    |       background_ready = 0
    |       global move_p = background_pose
    |       wv_wp2 = th_wv_wp2
    |       if(par_2f):
    |         background_cal=1
    |       else:
    |         background_cal=1
    |       end
    |       global a_val = 3
    |       if(a_val >= 30):
    |         write_port_register(142,112)
    |         sleep(0.5)
    |         halt
    |       end
    |     end
    | 
    |     if(wv_weldpar[5] ==1):
    |         if( (sin_dir==1 and wving_delay[0]==0) or (sin_dir==-1 and wving_delay[2]==0)):
    |          tri_count = tri_count + 1
    |         end
    |         global target_p = move_p[tri_count]
    |         target_p=p[target_p[0],target_p[1],target_p[2],target_p[3],target_p[4],target_p[5]]
    |         tri_count = tri_count + 1
    |     elif(wv_weldpar[5] ==2):
    |       if( (tri_count==1 and sin_dir==1 and wving_delay[0]==0) or (tri_count==1 and sin_dir==-1 and wving_delay[2]==0)):
    |        tri_count = tri_count + 1
    |       end
    |       global target_p = move_p[tri_count]
    |       target_p=p[target_p[0],target_p[1],target_p[2],target_p[3],target_p[4],target_p[5]]
    |       tri_count = tri_count + 1
    |     else:
    |       popup("Please insert 0 - sin or 1 - triangle")
    |     end
    |     if(target_p == p[0,0,0,0,0,0]):
    |       target_p = get_actual_tcp_pose()
    |     end
    |     # write_output_float_register(25,tri_count)
    |     if((norm(tri_count)== 1) and sin_dir==1 and wving_delay[0]>0):
    |       movel(target_p,a=a_val,v=wv_system_speed/1000)
    |       peak_value = 0
    |       sleep(wving_delay[0])
    |       peak_value = 100
    |     elif((norm(tri_count)== 2) and sin_dir==1 and wving_delay[1]>0):
    |       movel(target_p,a=a_val,v=wv_system_speed/1000)
    |       peak_value = 0
    |       sleep(wving_delay[1])
    |       peak_value = 100
    |     elif((norm(tri_count)== 1) and sin_dir==-1 and wving_delay[2]>0):
    |       movel(target_p,a=a_val,v=wv_system_speed/1000)
    |       peak_value = 0
    |       sleep(wving_delay[2])
    |       peak_value = 100
    |     elif((norm(tri_count)== 2) and sin_dir==-1 and wving_delay[3]>0):
    |       movel(target_p,a=a_val,v=wv_system_speed/1000)
    |       peak_value = 0
    |       sleep(wving_delay[3])
    |       peak_value = 100
    |     else:
    |       movel(target_p,a=a_val,v=wv_system_speed/1000)
    |       peak_value = 100
    |     end
    |     global last_pose = target_p
    |   end
    |   timer_1_is_counting = False
    | 
    |   if(a9_wv_weldingon == True and wving_crater[5]!=0):
    |     #crater end option
    |     set_current_voltage(wving_crater[3],wving_crater[4])
    |     sleep(wving_crater[5])
    |     program_weld_on = False
    |     set_current_voltage(ext_fun[1],ext_fun[0])
    |     if(isHicomm):
    |       write_port_register(202,0)
    |       write_port_register(149,0)
    |     else:
    |       set_standard_digital_out(0,False)
    |     end
    |     while(read_welder(5)==True):
    |       if(weld_onoff==True):
    |         write_welder(0,False)
    |       end
    |       sync()
    |     end
    |   end
    |   timer_counter = 0
    |   kill CThread
    |   kill DThread
    |   kill TThread
    |   timer_counter = 0
    |   timer_counting = False
    |   wcr_counter = 0
    |   wcr_counting = False
    |   get_wcr = False
    |   welding_off_t = 0
    | 
    |   if(wv_seq[0] == 0 or wv_seq[0] == 3):
    |     if(a9_wv_weldingon==True):
    |       program_weld_on = False
    |       write_port_register(202,0)
    |       write_port_register(149,0)
    |       write_welder(0,False)
    |       if(wv_weldpar[2]==1):
    |         target_pos = feature_offset(get_actual_tcp_pose(),p[0,0,-0.01,0,0,0],wv_Line_Feature2)
    |         movel(target_pos,0.5,0.01)
    |       end
    |     end
    |   end
    |   background_pose = [dumy_p,dumy_p,dumy_p]
    |   move_p = background_pose
    |   return sin_dir
    | end
    | 
    | 
    | def line_weaving_tp_l(wv_wp1,wv_wp3,wv_weldpar=[100,10,0,1,5,1,1],tilt_deg=[0,0,0],wving_delay=[0,0,0,0],welding_on=False,Arc_sen=[0,0,0,0,0,0],wv_gap=[0,0,0,0],z_param=[0,0,0,0,0],par_2f=False,wving_crater=[0,0,0,0,0,0,0,0,0,0],ext_fun=[0,0,0,0,0,0,0,0,0,0,0],wv_seq = [0,-1],wv_feature=p[0,0,0,0,0,0]):
    |   global start_gas_time = 2
    |   global counter_average = 1
    |   global counter_average_num = 0
    |   global waste_cycle = ext_fun[8]
    |   global current_list = 0
    |   global wv_wp4 = wv_wp3
    |   global A_T1 = wv_wp4[0]
    |   global A_T2 = wv_wp4[1]
    |   global A_T3 = wv_wp4[2]
    |   if(par_2f):
    |     global squash_cycle = 0
    |   else:
    |     global squash_cycle = ext_fun[7]
    |   end
    |   global th_ext_fun = ext_fun
    |   RTDE_init()
    | 
    |   if (wv_gap[0]==1):
    |     gap_check = True
    |     wv_gap[0]=0
    |   else:
    |     gap_check= False
    |   end
    |   # e-Series 2, CB-Seris 8
    |   global system_bus_ms = 2
    | 
    |   global sin_dir = wv_seq[1]
    |   global start_trig = False
    |   dir=1
    | 
    |   global tri_count=0
    | 
    |   global z_bottom = z_param[0]/1000
    |   if(wv_weldpar[6]==-1):
    |     global vir_v = -1
    |   else:
    |     global vir_v = 1
    |   end
    | 
    |   if(par_2f):
    |     global cal_off_ang_rx = 1
    |     global cal_off_ang_ry = 0
    |   else:
    |     global cal_off_ang_rx = 0
    |     global cal_off_ang_ry = 1
    |   end
    | 
    |   if(wv_seq[0] == 2 or wv_seq[0] == 3):
    |     tilt_deg = [0,0,0]
    |     global cal_off_ang_rx = 0
    |     global cal_off_ang_ry = 0
    |   end
    | 
    |   global wv_Line_Feature2 = wv_wp1
    |   if(wv_weldpar[0] > 700 and par_2f == False):
    |     wv_weldpar[0] = 700
    |   end
    |   if(wv_wp3[0]==p[0,0,0,0,0,0]):
    |     global wv_wp2 = feature_offset(wv_wp1,p[wv_weldpar[0]/1000,0,0,0,0,0],wv_Line_Feature2)
    |   else:
    |     global wv_wp2 = wv_wp4[0]
    |     wv_weldpar[0] = point_dist(wv_wp1,wv_wp2)*1000
    |     global wv_dist_bak = point_dist(wv_wp1,wv_wp2)*1000
    |   end
    |   if(wv_seq[0] == 2 or wv_seq[0] == 3):
    |     wv_Line_Feature2 = wv_feature
    |   end
    |   #setting
    |   if(par_2f):
    |     #todo - 1
    |     offset_2f_k = -1 * ext_fun[9]
    |     offset_2f_z = 1 * ext_fun[10]
    |     if(wv_seq[0] == 0 or wv_seq[0] == 1):
    |       line_feature = get_feature_Line(wv_wp1,wv_wp2)
    |       b_p1 = wv_wp1
    |       b_p2 = feature_offset(wv_wp1,p[0,0.01*vir_v,0,0,0,0],line_feature)
    |       b_p3 = pose_add(wv_wp1,p[0,0,0.01,0,0,0])
    | 
    |       back_feature = get_feature_plane_xz(b_p1,b_p2,b_p3)
    |       wv_wp1 = pose_trans(wv_wp1,p[0,0,0,0,0,d2r(-90)])
    |       wv_wp1 = feature_offset(wv_wp1,p[0,offset_2f_k/1000,0,0,0,0],back_feature)
    |       wv_wp1 = pose_add(wv_wp1,p[0,0,offset_2f_z/1000,0,0,0])
    |       # wv_wp1 = pose_add(wv_wp1,p[offset_2f_k/1000,0,0,0,0,0])
    |     end
    |       # wv_wp2 = pose_add(wv_wp2,p[offset_2f_k/1000,0,0,0,0,0])
    |       wv_wp2 = feature_offset(wv_wp2,p[0,offset_2f_k/1000,0,0,0,0],back_feature)
    |       wv_wp2 = pose_add(wv_wp2,p[0,0,offset_2f_z/1000,0,0,0])
    |       wv_wp2 = p[wv_wp2[0],wv_wp2[1],wv_wp2[2],wv_wp1[3],wv_wp1[4],wv_wp1[5]]
    | 
    |       wv_wp3_p = feature_offset(wv_wp3[0],p[0,offset_2f_k/1000,0,0,0,0],back_feature)
    |       wv_wp3_p = pose_add(wv_wp3_p,p[0,0,offset_2f_z/1000,0,0,0])
    |       wv_wp3_p = p[wv_wp3_p[0],wv_wp3_p[1],wv_wp3_p[2],wv_wp1[3],wv_wp1[4],wv_wp1[5]]
    |       wv_wp4[0] = p[wv_wp3_p[0],wv_wp3_p[1],wv_wp3_p[2],wv_wp1[3],wv_wp1[4],wv_wp1[5]]
    | 
    |       wv_wp3_p = feature_offset(wv_wp3[1],p[0,offset_2f_k/1000,0,0,0,0],back_feature)
    |       wv_wp3_p = pose_add(wv_wp3_p,p[0,0,offset_2f_z/1000,0,0,0])
    |       wv_wp3_p = p[wv_wp3_p[0],wv_wp3_p[1],wv_wp3_p[2],wv_wp1[3],wv_wp1[4],wv_wp1[5]]
    |       wv_wp4[1] = p[wv_wp3_p[0],wv_wp3_p[1],wv_wp3_p[2],wv_wp1[3],wv_wp1[4],wv_wp1[5]]
    | 
    |       wv_wp3_p = feature_offset(wv_wp3[2],p[0,offset_2f_k/1000,0,0,0,0],back_feature)
    |       wv_wp3_p = pose_add(wv_wp3_p,p[0,0,offset_2f_z/1000,0,0,0])
    |       wv_wp3_p = p[wv_wp3_p[0],wv_wp3_p[1],wv_wp3_p[2],wv_wp1[3],wv_wp1[4],wv_wp1[5]]
    |       wv_wp4[2] = p[wv_wp3_p[0],wv_wp3_p[1],wv_wp3_p[2],wv_wp1[3],wv_wp1[4],wv_wp1[5]]
    |   end
    |   if(ext_fun[2]==1 and par_2f==False):
    |     #squash
    |     w_voltage = ext_fun[3]
    |     w_current = ext_fun[4]
    |     set_current_voltage(w_current,w_voltage)
    |     global cir_speed_org_bak = wv_weldpar[1]
    |     global wving_amplitude_bak = wv_weldpar[4]
    |     wv_weldpar[1] = ext_fun[6]
    |     wv_weldpar[4] = ext_fun[5]
    |   end
    |   if(par_2f):
    |     global wv_system_speed = calculate_2f(wv_weldpar[4],wv_wp1,wv_wp2,wv_weldpar[1],wv_weldpar[3],wving_delay,wving_crater)
    |   else:
    |     global wv_system_speed = calculate_3f(wv_weldpar[4],wv_wp1,wv_wp2,wv_weldpar[1],wv_weldpar[3],wving_delay)
    |     x_radius = x_radius / 1000
    |   end
    |   global wv_set_speed = wv_system_speed
    |   ratio_t=0
    |   # mm -> m
    |   global y_radius = y_radius / 1000
    |   global y_radius_bak = y_radius
    |   #init for thread
    |   global ext_stick = 0
    |   global th_arc_sen=Arc_sen
    |   global th_wv_gap=wv_gap
    |   global th_tilt_deg=tilt_deg
    |   global last_tilt_deg =th_tilt_deg
    |   global last_wv_wp1 = wv_wp1
    |   global last_wv_line = wv_Line_Feature2
    |   global th_wving_crater=wving_crater
    |   global last_z_bottom = z_bottom
    |   global th_par_2f = par_2f
    |   global th_cir_speed_org=wv_weldpar[1]
    |   global th_wv_wp1 = wv_wp1
    |   global th_wv_wp2 = wv_wp2
    |   global th_wv_wp3 = wv_wp3[0]
    |   global th_wv_weldpar=wv_weldpar
    |   global th_wving_delay=wving_delay
    |   global th_z_param=z_param
    |   global th_wv_seq = wv_seq
    |   global th_wv_feature=wv_feature
    |   global th_dir = dir
    | 
    |   # if want to use approach position
    |   if(wv_seq[0] ==0 or wv_seq[0] == 1):
    |     global get_angle_rx = welding_angle_cal_2f(wv_wp1[1],tilt_deg,vir_v,cal_off_ang_rx)
    |     global get_angle_ry = welding_angle_cal_3f(wv_wp1[2],tilt_deg,z_bottom,cal_off_ang_ry)
    | 
    |     target_p = feature_offset(wv_wp1,p[0,0,0,d2r(tilt_deg[0] + get_angle_rx),d2r(tilt_deg[1] + get_angle_ry),d2r(tilt_deg[2])],wv_Line_Feature2)
    | 
    |     if(wv_weldpar[2]==1):
    |       target_p_appr = feature_offset(target_p,p[0,0,-0.02,0,0,0],wv_Line_Feature2)
    |       movel(target_p_appr,a=0.5,v=0.125)
    |     end
    |     movel(target_p,a=0.5,v=0.125)
    |   end
    | 
    |   CThread = run CalThread()
    |   DThread = run diff_Thread()
    |   TThread = run thread_timer()
    |   global timer_counting=True
    |   global program_weld_on = True
    | 
    |   if(a9_wv_weldingon==True):
    |     while(welding_off_t==55):
    |       sync()
    |     end
    |     if(wving_crater[2]>0):
    |       set_current_voltage(wving_crater[0],wving_crater[1])
    |     end
    |     if(welding_off_t != 1):
    |       write_welder(0,True)
    |       while(get_wcr==False):
    |         if(weld_onoff==False):
    |           write_welder(0,True)
    |         end
    |         sync()
    |       end
    |       if(wving_crater[2]>0):
    |         #Crater Begin option
    |         write_output_float_register(1,1)
    |         sleep(wving_crater[2])
    |         set_current_voltage(ext_fun[1],ext_fun[0])
    |       end
    |     end
    |   end
    |   start_gas_time = 0
    | 
    |   background_cal=1
    |   background_ready=0
    |   FT_trig=True
    | 
    |   timer_1_is_counting = True
    | 
    |   while((ratio_t < 1) or current_list==0 or current_list==1):
    |     if(ratio_t>=1 and current_list!=2):
    |       if (gap_check):
    |         gap_check = True
    |         wv_gap[0]=1
    |         th_wv_gap[0]=1
    |         gap_check= False
    |       end
    |       ratio_t=0
    |       if(current_list==0):
    |         wving_amp_bak = wv_weldpar[4]
    |         wv_weldpar[4] = wv_weldpar[4] * 1
    |         th_wv_weldpar[4] = wv_weldpar[4]
    |         circle_speed_bak = wv_weldpar[1]
    |         wv_weldpar[1]= wv_weldpar[1]*0.7
    |         th_wv_weldpar[1]= wv_weldpar[1]
    |       elif(current_list==1):
    |         wv_weldpar[4] = wving_amp_bak
    |         th_wv_weldpar[4] = wv_weldpar[4]
    |         wv_weldpar[1] = circle_speed_bak
    |         th_wv_weldpar[1]= wv_weldpar[1]
    |       end
    |       wv_wp1=wv_wp4[current_list]
    |       wv_wp2=wv_wp4[current_list+1]
    |       global th_wv_wp1 = wv_wp4[current_list]
    |       global th_wv_wp2 = wv_wp4[current_list+1]
    |       global th_wv_wp3 = wv_wp4[current_list+1]
    |       wv_system_speed_bak = wv_system_speed
    |       if(par_2f):
    |         global wv_system_speed = calculate_2f(wv_weldpar[4],wv_wp4[current_list],wv_wp4[current_list+1],wv_weldpar[1],wv_weldpar[3],wving_delay,wving_crater)
    |         global y_radius = y_radius / 1000
    |         global y_radius_bak = y_radius
    |       else:
    |         global wv_system_speed = calculate_3f(wv_weldpar[4],wv_wp4[current_list],wv_wp4[current_list+1],wv_weldpar[1],wv_weldpar[3],wving_delay)
    |         x_radius = x_radius / 1000
    |       end
    |       wv_system_speed = wv_system_speed_bak
    |       current_list=current_list+1
    |     end
    |     if((norm(tri_count)>=2 or (FT_trig==True))):
    |       FT_trig = False
    |       while(background_ready==0):
    |         sync()
    |       end
    |       tri_count = 0
    |       background_ready = 0
    |       global move_p = background_pose
    |       wv_wp2 = th_wv_wp2
    |       if(par_2f):
    |         background_cal=1
    |       else:
    |         background_cal=1
    |       end
    |       global a_val = 3
    |       if(a_val >= 30):
    |         write_port_register(142,112)
    |         sleep(0.5)
    |         halt
    |       end
    |     end
    | 
    |     if(wv_weldpar[5] ==1):
    |         if( (sin_dir==1 and wving_delay[0]==0) or (sin_dir==-1 and wving_delay[2]==0)):
    |          tri_count = tri_count + 1
    |         end
    |         global target_p = move_p[tri_count]
    |         target_p=p[target_p[0],target_p[1],target_p[2],target_p[3],target_p[4],target_p[5]]
    |         tri_count = tri_count + 1
    |     elif(wv_weldpar[5] ==2):
    |       if( (tri_count==1 and sin_dir==1 and wving_delay[0]==0) or (tri_count==1 and sin_dir==-1 and wving_delay[2]==0)):
    |        tri_count = tri_count + 1
    |       end
    |       global target_p = move_p[tri_count]
    |       target_p=p[target_p[0],target_p[1],target_p[2],target_p[3],target_p[4],target_p[5]]
    |       tri_count = tri_count + 1
    |     else:
    |       popup("Please insert 0 - sin or 1 - triangle")
    |     end
    | 
    |     if(target_p == p[0,0,0,0,0,0]):
    |       target_p = get_actual_tcp_pose()
    |     end
    |     if((norm(tri_count)== 1) and sin_dir==1 and wving_delay[0]>0):
    |       movel(target_p,a=a_val,v=wv_system_speed/1000)
    |       sleep(wving_delay[0])
    |     elif((norm(tri_count)== 2) and sin_dir==1 and wving_delay[1]>0):
    |       movel(target_p,a=a_val,v=wv_system_speed/1000)
    |       peak_value = 0
    |       sleep(wving_delay[1])
    |       peak_value = 100
    |     elif((norm(tri_count)== 1) and sin_dir==-1 and wving_delay[2]>0):
    |       movel(target_p,a=a_val,v=wv_system_speed/1000)
    |       sleep(wving_delay[2])
    |     elif((norm(tri_count)== 2) and sin_dir==-1 and wving_delay[3]>0):
    |       movel(target_p,a=a_val,v=wv_system_speed/1000)
    |       peak_value = 0
    |       sleep(wving_delay[3])
    |       peak_value = 100
    |     else:
    |       movel(target_p,a=a_val,v=wv_system_speed/1000)
    |     end
    |     global last_pose = target_p
    |   end
    |   timer_1_is_counting = False
    |   welding_program = True
    |   if(a9_wv_weldingon == True and wving_crater[5]!=0):
    |     #crater end option
    |     set_current_voltage(wving_crater[3],wving_crater[4])
    |     sleep(wving_crater[5])
    |     program_weld_on = False
    |     set_current_voltage(ext_fun[1],ext_fun[0])
    |     if(isHicomm):
    |       write_port_register(202,0)
    |       write_port_register(149,0)
    |     else:
    |       set_standard_digital_out(0,False)
    |     end
    |     while(get_wcr==True):
    |       if(weld_onoff==True):
    |         if(isHicomm):
    |           write_port_register(202,0)
    |           write_port_register(149,0)
    |         else:
    |           set_standard_digital_out(0,False)
    |         end
    |       end
    |       sync()
    |     end
    |   end
    | 
    |   kill CThread
    |   kill DThread
    |   kill TThread
    |   timer_counting = False
    |   wcr_counter = 0
    |   wcr_counting = False
    |   get_wcr = False
    |   welding_off_t = 0
    | 
    |   if(wv_seq[0] == 0 or wv_seq[0] == 3):
    |     if(a9_wv_weldingon==True):
    |       program_weld_on = False
    |       if(isHicomm):
    |         write_port_register(202,0)
    |         write_port_register(149,0)
    |       else:
    |         set_standard_digital_out(0,False)
    |       end
    |       if(wv_weldpar[2]==1):
    |         target_pos = feature_offset(get_actual_tcp_pose(),p[0,0,-0.01,0,0,0],wv_Line_Feature2)
    |         movel(target_pos,0.5,0.01)
    |       end
    |     end
    |   end
    |   background_pose = [dumy_p,dumy_p,dumy_p]
    |   move_p = background_pose
    |   return sin_dir
    | end
  Folder Reset [hidden by the author, left out]
  Folder Welding_Init [hidden by the author, left out]
  Folder init_reset_modbus_server [hidden by the author, left out]
Robot Program (runOnlyOnce=false)
  SuppressedNode
    Folder Folder [hidden by the author, left out]
  If simulation_mode
    'work mode 2'
    Script: write_port_register(162,2)
    touch_temp := 0
  If a0_Job_Mode≟1
    Folder job mode 1
      'JOB_MANUAL'
      Script: write_port_register(robot_ready_141,1)
      If freedrive≟ True  and freedrive_trg≟ False
        freedrive_trg := True
        Script: freedrive_mode()
      ElseIf freedrive≟ False  and freedrive_trg≟ True
        Script: end_freedrive_mode()
        freedrive_trg := False
      SuppressedNode
        If tool_in[0]≟ True  and Inch_trg≟ False removedSiblings(If(type=ElseIf checkContinuously=false, expression=tool_in[0]≟ False  and Inch_trg≟ True, children(Script(type=Line, expression=write_port_register(202,0)), Assignment(valueSource=Expression, variable=Inch_trg, expression=False))))
          Script: write_port_register(202,2)
          Inch_trg := True
      If freedrive≟ True  and save_tool≟ True
        SuppressedNode
          If freedrive_trg
            Script: end_freedrive_mode()
            freedrive_trg := False
        Wait Sleep waitTime=0.01
      ElseIf a1_job_move≟1
        'Manual - Move Home/Packing/Warmup'
        If read_port_register(robot_pose_164)≟1
          Script: write_port_register(robot_ready_141,0)
          Script: homeing()
          MoveJ speed 55 deg/s, acceleration 55 deg/s^2 (useActiveTCP=false)
            Waypoint Packing_pos referenceName=Packing_pos: TCP in base x=278.715 y=357.008 z=25.408 mm, rx=-2.147 ry=0.196 rz=-0.9199 rad; joints [90.973, -0.994, -143.143, -80.591, 93.211, 172.86] deg; flange x=104.677 y=49.288 z=284.06 mm, rx=0.249 ry=-2.8771 rz=-1.2051 rad
        ElseIf read_port_register(robot_pose_164)≟2
          Script: write_port_register(robot_ready_141,0)
          Script: homeing()
        ElseIf read_port_register(robot_pose_164)≟3 (checkContinuously=true)
          Script: write_port_register(robot_ready_141,0)
          Folder Warm-up [hidden by the author, left out]
          Script: homeing()
          Wait Sleep waitTime=2
        ElseIf read_port_register(robot_pose_164)≟4
          Script: write_port_register(robot_ready_141,0)
          Script: homeing()
          MoveJ speed 45 deg/s, acceleration 45 deg/s^2 (useActiveTCP=false)
            Waypoint pre_mounting: TCP in base x=460.443 y=114.922 z=277.199 mm, rx=-2.2401 ry=0.0674 rz=-1.6141 rad; joints [70.799, -49.866, -53.986, -136.967, 75.724, 151.917] deg; flange x=126.614 y=-35.489 z=517.648 mm, rx=-0.134 ry=2.6709 rz=0.506 rad
            Waypoint Mounting_pos: TCP in base x=365.658 y=-3.207 z=718.667 mm, rx=-1.2208 ry=-0.0667 rz=-2.3634 rad; joints [35.703, -36.102, -51.763, -101.417, 81.218, 101.941] deg; flange x=-17.293 y=-164.814 z=580.418 mm, rx=-0.2591 ry=1.737 rz=0.4847 rad
        ElseIf read_port_register(robot_pose_164)≟5
          c_p := get_actual_tcp_pose()
          MoveL speed 30 mm/s, acceleration 30 mm/s^2 (useActiveTCP=true) feature=Base
            m_p := pose_trans(c_p, p[0,0,0,d2r(tilt_deg_man),0,0])
            Waypoint Waypoint (Variable): variable=m_p
            m_p := pose_trans(c_p, p[0,0,0,d2r(-tilt_deg_man),0,0])
            Waypoint Waypoint (Variable): variable=m_p
            Waypoint Waypoint (Variable): variable=c_p
            m_p := pose_trans(c_p, p[0,0,0,0,d2r(tilt_deg_man),0])
            Waypoint Waypoint (Variable): variable=m_p
            m_p := pose_trans(c_p, p[0,0,0,0,d2r(-tilt_deg_man),0])
            Waypoint Waypoint (Variable): variable=m_p
            Waypoint Waypoint (Variable): variable=c_p
            m_p := pose_trans(c_p, p[0,0,0,0,0,d2r(tilt_deg_man)])
            Waypoint Waypoint (Variable): variable=m_p
            m_p := pose_trans(c_p, p[0,0,0,0,0,d2r(-tilt_deg_man)])
            Waypoint Waypoint (Variable): variable=m_p
            Waypoint Waypoint (Variable): variable=c_p
        Call Move_done
    Call robotand_cell_initalizat
  ElseIf a0_Job_Mode≟2 (checkContinuously=true)
    'JOB_AUTO'
    auto_on := True
    Folder Init [hidden by the author, left out]
    Folder Cell_calculation
      'setting'
      Auto_trig := False
      If Auto_trig≟ False
        If simulation_mode
          b1_cell_info_L := B
          b1_cell_info_R := B
          b1_cell_select := motion_num([A_VL1,A_VR1,A_HOR,0,0,0])
          b1_cell_select := motion_num([A_HOR,0,0,0,0,0])
          EXT_flag1 := integer_to_binary_list(read_port_register(2048))
          b1_cell_thickne := 6
          A_Touch_trig_l := touch_cal(b1_cell_info_L,b1_cell_info_R,b1_cell_select)
          Auto_W_num := cell_motion(A_Touch_trig_l,b1_cell_thickne,EXT_flag1,b1_cell_info_L,b1_cell_info_R)
          SuppressedNode
            Auto_W_num := cell_motion(b1_cell_select)
          Auto_total_cell := cell_num(Auto_W_num)
          Auto_trig := True
          A_sel_v := Auto_W_num[0]
        Else 
          b1_cell_info_L := read_port_register(171)
          b1_cell_info_R := read_port_register(172)
          EXT_flag1 := integer_to_binary_list(read_port_register(179))
          b1_cell_select := read_port_register(178)
          b1_cell_thickne := read_port_register(183)
          A_Touch_trig_l := touch_cal(b1_cell_info_L,b1_cell_info_R,b1_cell_select)
          Auto_W_num := cell_motion(A_Touch_trig_l,b1_cell_thickne,EXT_flag1,b1_cell_info_L,b1_cell_info_R)
          Auto_total_cell := cell_num(Auto_W_num)
          Auto_trig := True
          A_sel_v := Auto_W_num[0]
        Script: write_port_register(139,Auto_total_cell-1)
    Auto_cur_cell := 0
    Folder Touch,Welding
      'Calculate total sequence and decide way'
      Folder Calculate & Move & Touch
        Folder touch_init [hidden by the author, left out]
        If touch_temp≟0
          Script: write_port_register(138,0)
          Folder get_touch_position
            Folder get pre-positions
              If read_port_register(work_type_165)≟2
                Folder freedrive touch [hidden by the author, left out]
              Else 
                Folder value from pendant
                  move_i := 1
                  SuppressedNode
                    calcu_trig := True
                  Folder Touch_FrontandSide [hidden by the author, left out]
                  SuppressedNode
                    Wait Condition expression=calcu_trig≟ False
                  Wait Condition expression=event_side_on≟ False
            Folder move and touch
              Folder Touch Move
                Folder HOR_L [hidden by the author, left out]
                Folder VL1
                  If A_Prepos_l[A_VL1]≠p[0,0,0,0,0,0]
                    b2_left_par := True
                    b8_wv_2f := False
                    b7_tilt_degree := [0,0,0]
                    A_sel_v := A_VL1
                    A_sel_v_end := A_VL1_END
                    b2_par_cd := 0
                    If b1_cell_info_L≟A or b1_cell_info_L≟C or b1_cell_info_L≟c
                      Scallup_check := True
                    Else 
                      Scallup_check := False
                    Call MoveandTouchFun_3f
                    If b1_cell_info_L≟A or b1_cell_info_L≟C or b1_cell_info_L≟c
                      If A_Prepos_l[A_HOR]≟p[0,0,0,0,0,0]
                        Script: direction(p[0,0,0,0,0,0],[0,-1,0],8,120,160)
                        SuppressedNode
                          var_3 := get_actual_tcp_pose()
                        AAgcp := get_actual_tcp_pose()
                        AAgangle := up_left
                        AAgtp := p[AAgcp[0],AAgcp[1],AAgcp[2],AAgangle[3],AAgangle[4],AAgangle[5]]
                        MoveL speed 80 mm/s, acceleration 80 mm/s^2 (useActiveTCP=true) feature=Base
                          Waypoint Waypoint (Variable): variable(name=AAgtp)
                        SuppressedNode
                          Script: ori_move(var_3,up_left)
                        for_z_VL1 := contact_fun(p[0,0,0,0,0,0],[0,0,-1],10000,15,15,  False)
                        Script: direction(p[0,0,0,0,0,0],[0,0,1],20,120,160)
                        Script: write_welder(4, False )
                      Else 
                        for_z_VL1 := p[0,0,0,0,0,0]
                Folder HOR_ML [hidden by the author, left out]
                Folder VL2
                  If A_Prepos_l[A_VL2]≠p[0,0,0,0,0,0]
                    b2_left_par := True
                    b8_wv_2f := False
                    b7_tilt_degree := basic_tilt_3f
                    A_sel_v := A_VL2
                    A_sel_v_end := A_VL2_END
                    b2_par_cd := 1
                    If b1_cell_info_L≟A or b1_cell_info_L≟C or b1_cell_info_L≟c
                      Scallup_check := True
                    Else 
                      Scallup_check := False
                    If b1_cell_info_L≟d or b1_cell_info_L≟c
                      Halt
                    Else 
                      If A_Touch_p[A_VL1]≟p[0,0,0,0,0,0]
                        Call MoveandTouchFun_3f
                        If A_Prepos_l[A_HOR_ML]≟p[0,0,0,0,0,0]
                          Script: direction(p[0,0,0,0,0,0],[0,-1,0],8,120,160)
                          AAgcp := get_actual_tcp_pose()
                          AAgangle := up_left
                          AAgtp := p[AAgcp[0],AAgcp[1],AAgcp[2],AAgangle[3],AAgangle[4],AAgangle[5]]
                          MoveL speed 80 mm/s, acceleration 80 mm/s^2 (useActiveTCP=true) feature=Base
                            Waypoint Waypoint (Variable): variable=AAgtp
                          SuppressedNode
                            Script: ori_move(get_actual_tcp_pose(),up_left)
                          If b1_cell_info_L≠E and b1_cell_info_L≠e
                            for_cal_zl := contact_fun(p[0,0,0,0,0,0],[0,0,-1],20000,20,20)
                            Script: direction(p[0,0,0,0,0,0],[0,0,1],10,120,160)
                        touch_tmp := A_Touch_p[A_sel_v]
                        If b1_cell_info_L≠E and b1_cell_info_L≠e
                          Script: touch_tmp[2]=for_cal_zl[2]
                          Script: A_Touch_p[A_sel_v]=touch_tmp
                        for_cal_y_wel := A_Touch_p[A_sel_v]
                        for_cal_x_wel := A_Touch_p[A_sel_v]
                      Else 
                        Call MoveFun
                        for_cal_y_wel := contact_fun(p[0,0,0,0,0,0],[1,0,0],20000,20,20)
                        Script: direction(p[0,0,0,0,0,0],[-1,0,0],40,120,160)
                        If A_Prepos_l[A_HOR_ML]≟p[0,0,0,0,0,0]
                          Script: direction(p[0,0,0,0,0,0],[0,1,0],60,120,160)
                          var_2 := contact_fun(p[0,0,0,0,0,0],[1,0,0],20000,20,20)
                          Script: direction(p[0,0,0,0,0,0],[-1,0,0],5,120,160)
                          Script: direction(p[0,0,0,0,0,0],[0,-1,0],60,120,160)
                          Script: direction(p[0,0,0,0,0,0],[1,0,0],10,120,160)
                          for_cal_x_wel := contact_fun(p[0,0,0,0,0,0],[0,1,0],20000,20,20)
                          Script: direction(p[0,0,0,0,0,0],[0,-1,0],20,120,160)
                          AAgcp := get_actual_tcp_pose()
                          AAgangle := up_left
                          AAgtp := p[AAgcp[0],AAgcp[1],AAgcp[2],AAgangle[3],AAgangle[4],AAgangle[5]]
                          MoveL speed 80 mm/s, acceleration 80 mm/s^2 (useActiveTCP=true) feature=Base
                            Waypoint Waypoint (Variable): variable=AAgtp
                          SuppressedNode
                            Script: ori_move(get_actual_tcp_pose(),up_left)
                          If b1_cell_info_L≠E and b1_cell_info_L≠e
                            for_cal_zl := contact_fun(p[0,0,0,0,0,0],[0,0,-1],20000,20,20)
                            Script: direction(p[0,0,0,0,0,0],[0,0,1],10,120,160)
                          Script: direction(p[0,0,0,0,0,0],[-1,0,0],20,120,160)
                        for_cal_rot := A_Touch_p[A_VL1]
                        If b1_cell_info_L≠E and b1_cell_info_L≠e
                          Script: A_Touch_p[A_sel_v]=p[for_cal_y_wel[0],for_cal_x_wel[1],for_cal_zl[2],for_cal_rot[3],for_cal_rot[4],for_cal_rot[5]]
                          Script: touch_tmp=p[for_cal_y_wel[0],for_cal_x_wel[1],for_cal_zl[2],for_cal_rot[3],for_cal_rot[4],for_cal_rot[5]]
                        Else 
                          Script: touch_tmp=p[for_cal_y_wel[0],for_cal_x_wel[1],for_cal_x_wel[2],for_cal_rot[3],for_cal_rot[4],for_cal_rot[5]]
                        If Scallup_check≟ False
                          touch_tmp := pose_trans(touch_tmp,p[-(Touch_dis)/1000,0,0,0,0,0])
                          Script: A_Touch_p[A_sel_v]=touch_tmp
                        Else 
                          Scallup_check := False
                        Script: write_welder(4, False )
                    b2_par_cd := 0
                    Script: homeing()
                  Else 
                    Script: homeing()
                Folder HOR_R [hidden by the author, left out]
                Folder VR1 [hidden by the author, left out]
                Folder HOR_MR [hidden by the author, left out]
                Folder VR2
                  If A_Prepos_l[A_VR2]≠p[0,0,0,0,0,0]
                    Folder Init [hidden by the author, left out]
                    If b1_cell_info_R≟A or b1_cell_info_R≟C or b1_cell_info_R≟c
                      Scallup_check := True
                    Else 
                      Scallup_check := False
                    If b1_cell_info_R≟d or b1_cell_info_R≟c
                      If vr2_p1≟p[0,0,0,0,0,0]
                        Call MoveFun_cd
                        vr2_p1 := contact_fun(p[0,0,0,0,0,0],[1,0,0],20000,20,20)
                        Script: direction(p[0,0,0,0,0,0],[-1,0,0],20,120,160)
                        Script: direction(p[0,0,0,0,0,0],[0,1,0],10,120,160)
                        vr2_p2 := contact_fun(p[0,0,0,0,0,0],[1,0,0],20000,20,20)
                        Script: direction(p[0,0,0,0,0,0],[-1,0,0],14,120,160)
                        vr2_p3 := contact_fun(p[0,0,0,0,0,0],[0,1,0],20000,20,20)
                        Script: direction(p[0,0,0,0,0,0],[0,-1,0],30,120,160)
                        Script: direction(p[0,0,0,0,0,0],[-1,0,0],20,120,160)
                        vr2_p4 := contact_fun(p[0,0,0,0,0,0],[0,0,-1],20000,20,20)
                        Script: direction(p[0,0,0,0,0,0],[0,0,1],40,120,160)
                        Script: A_Touch_p[A_sel_v]=touch_xyz_get_middle(vr2_p1,vr2_p2,vr2_p3,vr2_p4)
                        var_4 := A_Touch_p[A_sel_v]
                        var_4 := pose_trans(var_4, p[a6_callar_vert/1000,0,0,0,0,0])
                        var_5 := get_actual_tcp_pose()
                        Script: var_5[2]=var_4[2]
                        var_5 := pose_trans(var_5, p[0,0,0,0,d2r(10),0])
                        MoveL speed 100 mm/s, acceleration 100 mm/s^2 (useActiveTCP=true) feature=Base
                          Waypoint Waypoint (Variable): variable=var_5
                        vr2_p1_up := contact_fun(p[0,0,0,0,0,0],[1,0,0],20000,20,20)
                        Script: direction(p[0,0,0,0,0,0],[-1,0,0],20,120,160)
                        Script: direction(p[0,0,0,0,0,0],[0,1,0],10,120,160)
                        vr2_p2_up := contact_fun(p[0,0,0,0,0,0],[1,0,0],20000,20,20)
                        Script: direction(p[0,0,0,0,0,0],[-1,0,0],14,120,160)
                        vr2_p3_up := contact_fun(p[0,0,0,0,0,0],[0,1,0],20000,20,20)
                        Script: direction(p[0,0,0,0,0,0],[0,-1,0],30,120,160)
                        Script: direction(p[0,0,0,0,0,0],[-1,0,0],20,120,160)
                      Script: A_Touch_p[A_sel_v+9]=touch_4point(vr2_p1_up,vr2_p2_up,vr2_p3_up)
                      Script: A_Touch_p[A_sel_v+9]=ori_pose(A_Touch_p[A_sel_v+9],A_Touch_p[A_sel_v])
                    Else 
                      If A_Touch_p[A_VR1]≟p[0,0,0,0,0,0]
                        Call MoveandTouchFun_3f
                        touch_tmp := A_Touch_p[A_sel_v]
                        If A_Prepos_l[A_HOR_MR]≟p[0,0,0,0,0,0]
                          Script: direction(p[0,0,0,0,0,0],[0,1,0],8,120,160)
                          AAgcp := get_actual_tcp_pose()
                          AAgangle := up_right
                          AAgtp := p[AAgcp[0],AAgcp[1],AAgcp[2],AAgangle[3],AAgangle[4],AAgangle[5]]
                          MoveL speed 80 mm/s, acceleration 80 mm/s^2 (useActiveTCP=true) feature=Base
                            Waypoint Waypoint (Variable): variable=AAgtp
                          SuppressedNode
                            Script: ori_move(get_actual_tcp_pose(),up_right)
                        If b1_cell_info_R≠E and b1_cell_info_R≠e
                          for_cal_zr := contact_fun(p[0,0,0,0,0,0],[0,0,-1],20000,20,20)
                          Script: touch_tmp[2]=for_cal_zr[2]
                        Script: A_Touch_p[A_sel_v]=touch_tmp
                        for_cal_y_wel := A_Touch_p[A_sel_v]
                        for_cal_x_wel := A_Touch_p[A_sel_v]
                      Else 
                        Call MoveFun
                        for_cal_y_wel := contact_fun(p[0,0,0,0,0,0],[1,0,0],20000,20,20)
                        Script: direction(p[0,0,0,0,0,0],[-1,0,0],40,120,160)
                        If A_Prepos_l[A_HOR_MR]≟p[0,0,0,0,0,0]
                          Script: direction(p[0,0,0,0,0,0],[0,-1,0],60,120,160)
                          var_2 := contact_fun(p[0,0,0,0,0,0],[1,0,0],20000,20,20)
                          Script: direction(p[0,0,0,0,0,0],[-1,0,0],5,120,160)
                          Script: direction(p[0,0,0,0,0,0],[0,1,0],60,120,160)
                          Script: direction(p[0,0,0,0,0,0],[1,0,0],10,120,160)
                          for_cal_x_wel := contact_fun(p[0,0,0,0,0,0],[0,-1,0],20000,20,20)
                          Script: direction(p[0,0,0,0,0,0],[0,1,0],20,120,160)
                          AAgcp := get_actual_tcp_pose()
                          AAgangle := up_right
                          AAgtp := p[AAgcp[0],AAgcp[1],AAgcp[2],AAgangle[3],AAgangle[4],AAgangle[5]]
                          MoveL speed 100 mm/s, acceleration 100 mm/s^2 (useActiveTCP=true) feature=Base
                            Waypoint Waypoint (Variable): variable=AAgtp
                          SuppressedNode
                            Script: ori_move(get_actual_tcp_pose(),up_right)
                          If b1_cell_info_R≠E and b1_cell_info_R≠e
                            for_cal_zr := contact_fun(p[0,0,0,0,0,0],[0,0,-1],20000,20,20)
                            Script: direction(p[0,0,0,0,0,0],[0,0,1],20,120,160)
                          Script: direction(p[0,0,0,0,0,0],[-1,0,0],20,120,160)
                        for_cal_rot := A_Touch_p[A_VR1]
                        If b1_cell_info_R≠E and b1_cell_info_R≠e
                          Script: A_Touch_p[A_sel_v]=p[for_cal_y_wel[0],for_cal_x_wel[1],for_cal_zr[2],for_cal_rot[3],for_cal_rot[4],for_cal_rot[5]]
                          Script: touch_tmp=p[for_cal_y_wel[0],for_cal_x_wel[1],for_cal_zr[2],for_cal_rot[3],for_cal_rot[4],for_cal_rot[5]]
                        Else 
                          Script: A_Touch_p[A_sel_v]=p[for_cal_y_wel[0],for_cal_x_wel[1],for_cal_x_wel[2],for_cal_rot[3],for_cal_rot[4],for_cal_rot[5]]
                          Script: touch_tmp=p[for_cal_y_wel[0],for_cal_x_wel[1],for_cal_x_wel[2],for_cal_rot[3],for_cal_rot[4],for_cal_rot[5]]
                        If Scallup_check≟ False
                          touch_tmp := pose_trans(touch_tmp,p[-(Touch_dis)/1000,0,0,0,0,0])
                          Script: A_Touch_p[A_sel_v]=touch_tmp
                        Else 
                          Scallup_check := False
                        Script: write_welder(4, False )
                    b2_par_cd := 0
                    Script: homeing()
                  Else 
                    Script: homeing()
                Script: write_welder(4,False)
                SuppressedNode
                  If A_Prepos_l[A_VR2]≠p[0,0,0,0,0,0] removedSiblings(If(type=Else checkContinuously=false, children(Script(type=Line, expression=homeing()))))
                    b2_left_par := False
                    b8_wv_2f := False
                    b7_tilt_degree := basic_tilt_3f
                    A_sel_v := A_VR2
                    A_sel_v_end := A_VR2_END
                    b2_par_cd := 1
                    If b1_cell_info_R≟A or b1_cell_info_R≟C or b1_cell_info_R≟c
                      Scallup_check := True
                    Else 
                      Scallup_check := False
                    If b1_cell_info_R≟d or b1_cell_info_R≟c
                      Halt
                    Else 
                      If A_Touch_p[A_VR1]≟p[0,0,0,0,0,0]
                        CallSubProgram
                        touch_tmp := A_Touch_p[A_sel_v]
                        If A_Prepos_l[A_HOR_MR]≟p[0,0,0,0,0,0]
                          Script: direction(p[0,0,0,0,0,0],[0,1,0],8,120,160)
                          AAgcp := get_actual_tcp_pose()
                          AAgangle := up_right
                          AAgtp := p[AAgcp[0],AAgcp[1],AAgcp[2],AAgangle[3],AAgangle[4],AAgangle[5]]
                          MoveL speed 250 mm/s, acceleration 1200 mm/s^2 (useActiveTCP=true) feature=Base
                            Waypoint Waypoint (Variable): variable=AAgtp
                          SuppressedNode
                            Script: ori_move(get_actual_tcp_pose(),up_right)
                          for_cal_zr := contact_fun(p[0,0,0,0,0,0],[0,0,-1],20000,20,20)
                        Script: touch_tmp[2]=for_cal_zr[2]
                        Script: A_Touch_p[A_sel_v]=touch_tmp
                        for_cal_y_wel := A_Touch_p[A_sel_v]
                        for_cal_x_wel := A_Touch_p[A_sel_v]
                      Else 
                        CallSubProgram
                        for_cal_y_wel := contact_fun(p[0,0,0,0,0,0],[1,0,0],20000,20,20)
                        Script: direction(p[0,0,0,0,0,0],[-1,0,0],40,120,160)
                        If A_Prepos_l[A_HOR_MR]≟p[0,0,0,0,0,0]
                          Script: direction(p[0,0,0,0,0,0],[0,-1,0],60,120,160)
                          var_2 := contact_fun(p[0,0,0,0,0,0],[1,0,0],20000,20,20)
                          Script: direction(p[0,0,0,0,0,0],[-1,0,0],5,120,160)
                          Script: direction(p[0,0,0,0,0,0],[0,1,0],60,120,160)
                          Script: direction(p[0,0,0,0,0,0],[1,0,0],10,120,160)
                          for_cal_x_wel := contact_fun(p[0,0,0,0,0,0],[0,-1,0],20000,20,20)
                          Script: direction(p[0,0,0,0,0,0],[0,1,0],20,120,160)
                          AAgcp := get_actual_tcp_pose()
                          AAgangle := up_right
                          AAgtp := p[AAgcp[0],AAgcp[1],AAgcp[2],AAgangle[3],AAgangle[4],AAgangle[5]]
                          MoveL speed 250 mm/s, acceleration 1200 mm/s^2 (useActiveTCP=true) feature=Base
                            Waypoint Waypoint (Variable): variable=AAgtp
                          SuppressedNode
                            Script: ori_move(get_actual_tcp_pose(),up_right)
                          for_cal_zr := contact_fun(p[0,0,0,0,0,0],[0,0,-1],20000,20,20)
                          Script: direction(p[0,0,0,0,0,0],[0,0,1],20,120,160)
                          Script: direction(p[0,0,0,0,0,0],[-1,0,0],20,120,160)
                        for_cal_rot := A_Touch_p[A_VR1]
                        Script: A_Touch_p[A_sel_v]=p[for_cal_y_wel[0],for_cal_x_wel[1],for_cal_zr[2],for_cal_rot[3],for_cal_rot[4],for_cal_rot[5]]
                        Script: write_welder(4, False )
                    b2_par_cd := 0
                    Script: homeing()
              Folder Touch After Offset
                Folder touch_after_offset
                  Folder HOR [hidden by the author, left out]
                  Folder VL1
                    If A_Prepos_l[A_VL1]≠p[0,0,0,0,0,0]
                      If b1_cell_info_L≟A or b1_cell_info_L≟C or b1_cell_info_L≟c
                        '3f only does not apply offset'
                        If for_z_VL1≟p[0,0,0,0,0,0]
                          for_z_VL1 := A_Touch_p[A_HOR]
                        ''
                        If for_z_VL1≠p[0,0,0,0,0,0]
                          z_diff := get_feature_pose(for_z_VL1,A_Touch_p[A_VL1])
                          Script: A_Touch_p[A_VL1]=pose_trans(A_Touch_p[A_VL1], p[z_diff[0],0,0,0,0,0])
                        SuppressedNode
                          Script: A_Touch_p[A_VL1]=put_pose(A_Touch_p[A_VL1],2, for_z_VL1[2])
                      Script: A_Touch_p[A_VL1]=pose_trans(A_Touch_p[A_VL1], p[offset_3f_begin/1000,0,0,0,0,0])
                  Folder VL2
                    If A_Prepos_l[A_VL2]≠p[0,0,0,0,0,0]
                      Script: A_Touch_p[A_VL2]=pose_trans(A_Touch_p[A_VL2], p[offset_3f_begin/1000,0,0,0,0,0])
                  Folder HOR_R
                    If A_Prepos_l[A_HOR_R]≠p[0,0,0,0,0,0]
                      If b1_cell_info_R≟A or b1_cell_info_R≟C or b1_cell_info_R≟c
                        If for_x_HOR_R≟p[0,0,0,0,0,0]
                          for_x_HOR_R := A_Touch_p[A_VR1]
                        If for_x_HOR≠p[0,0,0,0,0,0]
                          x_diff := get_feature_pose(for_x_HOR_R,A_Touch_p[A_HOR_R])
                          Script: A_Touch_p[A_HOR_R]=pose_trans(A_Touch_p[A_HOR_R], p[x_diff[0],0,0,0,0,0])
                      Script: A_Touch_p[A_HOR_R]=pose_trans(A_Touch_p[A_HOR_R], p[-offset_2f_begin/1000,0,0,0,0,0])
                  Folder VR1 [hidden by the author, left out]
                  Folder VR2
                    If A_Prepos_l[A_VR2]≠p[0,0,0,0,0,0]
                      Script: A_Touch_p[A_VR2]=pose_trans(A_Touch_p[A_VR2], p[offset_3f_begin/1000,0,0,0,0,0])
                  Folder HOR_ML [hidden by the author, left out]
                  Folder HOR_MR [hidden by the author, left out]
              'Touch Remember On/OFF'
              Script: write_port_register(180,1)
        Else 
          Folder Ignore Touch and check error [hidden by the author, left out]
      Folder welding
        Folder weldings [hidden by the author, left out]
  Wait Sleep waitTime=0.01
  Folder after init auto
    If auto_on
      Script: write_port_register(202,0)
      Timer (action=Stop) variable=timer_1
      Script: write_welder(0, False )
      Script: write_welder(4, False )
      Call reset_weld_param
      multi_path := 1
      auto_on := False
      current_2f := 0
      get_center := get_center_bak
      vr2_p1 := p[0,0,0,0,0,0]
      welding_program := False
      start_num := 135
      Loop While (checkContinuously=false) expression=start_num<141
        Script: write_port_register(start_num,0)
        start_num := start_num+1
Thread Thread_2 (runOnlyOnce=false)
  heartbeat := heartbeat+1
  If heartbeat>499
    heartbeat := 0
  Script: write_port_register(128,heartbeat)
  SuppressedNode
    Folder Pendant_Heartbeat
      If pendant_hb≟read_port_register(161)
        pb_comm_count := pb_comm_count+1
      Else 
        pendant_hb := read_port_register(161)
        pb_comm_count := 0
      If pb_comm_count≥5
        Script: write_port_register(142,151)
        Halt
  Wait Sleep waitTime=1
Thread Thread_1 (runOnlyOnce=false)
  a0_Job_Mode := read_port_register(162)
  a1_job_move := read_port_register(163)
  If red_led≟ True
    Set DigitalOutput pin=red_led; digitalValue=0
  If a0_Job_Mode≟2
    If read_port_register(arc_onoff_168)≟2
      a9_wv_weldingon := True
    Else 
      a9_wv_weldingon := False
    If Auto_trig
      get_next_number := read_port_register(166)
      get_move_trig := read_port_register(167)
      If get_move_trig≟1 and running_trig≟ True
        If get_next_number<0 or get_next_number>30
          Script: write_port_register(142,141)
          Halt
        If get_next_number≠Auto_cur_cell
          running_trig := False
          Script: write_welder(0, False )
          Script: write_port_register(149,0)
          Script: write_port_register(202,0)
        Else 
          Script: write_port_register(166,0)
          Script: write_port_register(167,0)
    If t_time>timer_1
      Script: write_port_register(143,timer_1)
    Else 
      Script: write_port_register(143,timer_1)
      Script: write_port_register(144,timer_1)
    Folder Monitoring touch and welding [hidden by the author, left out]
  If get_tool_digital_in(1)≟ True
    Script: set_tool_digital_out(1, False )
  Else 
    Script: set_tool_digital_out(1, True )
  If red_led≟ True
    Set DigitalOutput pin=red_led; digitalValue=0
    Script: end_freedrive_mode()
  Script: check_speed()
  Wait Sleep waitTime=0.05
Event  expression=event_cal_on
  SuppressedNode
    A_Speed_list := [0, 0, 0, 0, 0, 0, 0, 0, 0, 0, 0, 0, 0, 0, 0, 0]
  SuppressedNode
    A_Distance_list := [0, 0, 0, 0, 0, 0, 0, 0, 0, 0, 0, 0, 0, 0, 0, 0]
  move_i_f := 1
  get_pose_side := 0
  Loop While (checkContinuously=false) expression=move_i_f<10
    If A_Touch_trig_l[move_i_f]≟ True
      If move_i_f≟A_VL1 or move_i_f≟A_VL2
        A_sel_v := move_i_f
        If simulation_mode
          Call welding_parameter_sim
        Else 
          Call welding_parameter_init
        If a8_wv_distance<5
          Script: write_port_register(142,143)
          Halt
        b2_left_par := True
        b8_wv_2f := False
        If move_i_f≟A_VL2
          callar_hor := a6_callar_hor
          b2_cell := 0
          If b1_cell_info_L≟c or b1_cell_info_L≟d or b1_cell_info_L≟E or b1_cell_info_L≟e
            b2_cell := b1_cell_info_L
          Else 
            b2_cell := 0
        Else 
          callar_hor := 0
          b2_cell := b1_cell_info_L
        get_pos := get_lr(left,a6_f_width,a5_f_hole,a7_f_distance,b2_left_par,b8_wv_2f,Touch_dis,get_margin_z,get_pose_side,callar_hor,b2_cell,center_line)
        pre_tp := tilt_3f_fun(get_pos,[0,0,0],0)
        Script: A_Prepos_l[move_i_f]=pre_tp
      ElseIf move_i_f≟A_VR1 or move_i_f≟A_VR2
        A_sel_v := move_i_f
        If simulation_mode
          Call welding_parameter_sim
        Else 
          Call welding_parameter_init
        If a8_wv_distance<5
          Script: write_port_register(142,143)
          Halt
        b2_left_par := False
        b8_wv_2f := False
        If move_i_f≟A_VR2
          callar_hor := a6_callar_hor
          If b1_cell_info_R≟c or b1_cell_info_R≟d or b1_cell_info_R≟E or b1_cell_info_R≟e
            b2_cell := b1_cell_info_R
          Else 
            b2_cell := 0
        Else 
          callar_hor := 0
          b2_cell := b1_cell_info_R
        get_pos := get_lr(right,a6_f_width,a5_f_hole,a7_f_distance,b2_left_par,b8_wv_2f,Touch_dis,get_margin_z,get_pose_side,callar_hor,b2_cell,center_line)
        pre_tp := tilt_3f_fun(get_pos,[0,0,0],0)
        Script: A_Prepos_l[move_i_f]=pre_tp
      ElseIf move_i_f≟A_HOR
        A_sel_v := A_HOR
        If simulation_mode
          Call welding_parameter_sim
        Else 
          Call welding_parameter_init
        b8_wv_2f := True
        b2_left_par := True
        b2_cell := b1_cell_info_L
        get_pos := get_lr(up_left,a6_f_width,a5_f_hole,a7_f_distance,b2_left_par,b8_wv_2f,Touch_dis,get_margin_z,get_pose_side,0,b2_cell,center_line)
        pre_tp := get_pos
        Script: A_Prepos_l[move_i_f]=pre_tp
      ElseIf move_i_f≟A_HOR_R
        A_sel_v := A_HOR
        If simulation_mode
          Call welding_parameter_sim
        Else 
          Call welding_parameter_init
        b2_left_par := False
        b8_wv_2f := True
        b2_cell := b1_cell_info_R
        get_pos := get_lr(up_right,a6_f_width,a5_f_hole,a7_f_distance,b2_left_par,b8_wv_2f,Touch_dis,get_margin_z,get_pose_side,0,b2_cell,center_line)
        pre_tp := get_pos
        Script: A_Prepos_l[move_i_f]=pre_tp
      ElseIf move_i_f≟A_HOR_ML
        A_sel_v := A_HOR_ML
        If simulation_mode
          Call welding_parameter_sim
        Else 
          Call welding_parameter_init
        b8_wv_2f := True
        b2_left_par := True
        b2_cell := b1_cell_info_L
        Touch_dis := -1*Touch_dis
        get_pos := get_lr(up_left,a6_f_width,a5_f_hole,a7_f_distance,b2_left_par,b8_wv_2f,Touch_dis,get_margin_z,get_pose_side,a6_callar_hor,b2_cell,center_line)
        Touch_dis := -1*Touch_dis
        pre_tp := get_pos
        Script: A_Prepos_l[move_i_f]=pre_tp
      ElseIf move_i_f≟A_HOR_MR
        A_sel_v := A_HOR_MR
        If simulation_mode
          Call welding_parameter_sim
        Else 
          Call welding_parameter_init
        b2_left_par := False
        b8_wv_2f := True
        b2_cell := b1_cell_info_R
        Touch_dis := -1*Touch_dis
        get_pos := get_lr(up_right,a6_f_width,a5_f_hole,a7_f_distance,b2_left_par,b8_wv_2f,Touch_dis,get_margin_z,get_pose_side,a6_callar_hor,b2_cell,center_line)
        Touch_dis := -1*Touch_dis
        pre_tp := get_pos
        Script: A_Prepos_l[move_i_f]=pre_tp
      If move_i_f≤4
        Script: A_Prepos_l[move_i_f+9]=p[0,0,0,0,0,0]
      SuppressedNode
        Script: A_Speed_list[move_i]=a2_speed_cpm
      SuppressedNode
        Script: A_Distance_list[move_i]=a8_wv_distance
    move_i_f := move_i_f+1
  event_cal_on := False
Event  expression=event_side_on
  SuppressedNode
    A_Speed_list := [0, 0, 0, 0, 0, 0, 0, 0, 0, 0, 0, 0, 0, 0, 0, 0]
  SuppressedNode
    A_Distance_list := [0, 0, 0, 0, 0, 0, 0, 0, 0, 0, 0, 0, 0, 0, 0, 0]
  Wait Condition expression=event_cal_on≟ False
  move_i_f := 1
  get_pose_side := get_pose_side_t
  Loop While (checkContinuously=false) expression=move_i_f<10
    If A_Touch_trig_l[move_i_f]≟ True
      If move_i_f≟A_VL1 or move_i_f≟A_VL2
        Script: A_Prepos_l[move_i_f]=side_apply(A_Prepos_l[move_i_f],center_line,get_pose_side)
      ElseIf move_i_f≟A_VR1 or move_i_f≟A_VR2
        Script: A_Prepos_l[move_i_f]=side_apply(A_Prepos_l[move_i_f],center_line,get_pose_side)
      ElseIf move_i_f≟A_HOR
        Script: A_Prepos_l[move_i_f]=side_apply(A_Prepos_l[move_i_f],center_line,get_pose_side)
      ElseIf move_i_f≟A_HOR_R
        Script: A_Prepos_l[move_i_f]=side_apply(A_Prepos_l[move_i_f],center_line,get_pose_side)
      ElseIf move_i_f≟A_HOR_ML
        Script: A_Prepos_l[move_i_f]=side_apply(A_Prepos_l[move_i_f],center_line,get_pose_side)
      ElseIf move_i_f≟A_HOR_MR
        Script: A_Prepos_l[move_i_f]=side_apply(A_Prepos_l[move_i_f],center_line,get_pose_side)
    move_i_f := move_i_f+1
  event_side_on := False
Event  expression=reset_trig
  Call reset_weld_param
  reset_trig := False
Event  expression=time_cal_trig
  t_time := time_cal(Auto_W_num,Auto_total_cell,A_Speed_list,A_Distance_list,A_Touch_p,0)
  Script: write_port_register(144,t_time)
  time_cal_trig := False
Event  expression=pause_trig
  s_conn := socket_open("192.168.1.7",29999)
  s_send := socket_send_string("pause")
  s_send := socket_send_byte(10)
  Script: socket_close()
  pause_trig := False
SubProgram  [hidden by the author, left out]
SubProgram  [hidden by the author, left out]
SubProgram -> welding_parameter_init
SubProgram  [hidden by the author, left out]
SubProgram  [hidden by the author, left out]
SubProgram  [hidden by the author, left out]
SubProgram  [hidden by the author, left out]
SubProgram  [hidden by the author, left out]
SubProgram -> MoveandTouchFun_3f
SubProgram  [hidden by the author, left out]
SubProgram -> weav_welding_2f
SubProgram -> weav_welding_2f_CD
SubProgram  [hidden by the author, left out]
SubProgram  [hidden by the author, left out]
SubProgram Move_done [hidden by the author, left out]
SubProgram MoveandTouchFun_3f (keepSynchronizedWithDisk=false)
  b_touch_pos := A_Prepos_l[A_sel_v]
  tilt_deg_ry := 0
  tilt_deg_rz := 0
  If b2_left_par
    tilt_deg := 6
    b_touch_pos := pose_trans(b_touch_pos, p[0,0/1000,0,d2r(tilt_deg),d2r(tilt_deg_ry),d2r(tilt_deg_rz)])
  Else 
    tilt_deg := 0.5
    b_touch_pos := pose_trans(b_touch_pos, p[0,0/1000,0,d2r(-tilt_deg),d2r(tilt_deg_ry),d2r(tilt_deg_rz)])
  SuppressedNode
    Folder old
      Folder Pre_pos
        If b2_left_par and b_touch_pos[1]>0.305
          MoveJ speed 60 deg/s, acceleration 80 deg/s^2 (useActiveTCP=true)
            Waypoint left_prep: TCP in base x=399.324 y=304.924 z=155.271 mm, rx=-2.012 ry=-1.0104 rz=-1.4456 rad; joints [58.353, -52.164, -91.55, -103.62, 84.819, 95.689] deg; flange x=171.612 y=49.86 z=428.405 mm, rx=-1.1979 ry=2.4763 rz=0.1792 rad
        ElseIf b2_left_par≟ False  and b_touch_pos[1]<-0.283
          MoveJ speed 60 deg/s, acceleration 80 deg/s^2 (useActiveTCP=true)
            Waypoint right_prep: TCP in base x=454.066 y=-283.902 z=116.638 mm, rx=2.2253 ry=-0.6942 rz=1.4835 rad; joints [20.297, -58.556, -92.591, -108.708, 71.582, 144.682] deg; flange x=195.53 y=-75.381 z=401.578 mm, rx=0.8644 ry=2.6591 rz=-0.2158 rad
      MoveL speed 250 mm/s, acceleration 1200 mm/s^2 (useActiveTCP=true) feature=Base
        Waypoint Waypoint (Variable): variable=b_touch_pos
  Folder move_pre
    If (b2_left_par≟ True  and point_dist(A_Prepos_l[A_HOR], A_Prepos_l[A_VL1])>0.03) or (b2_left_par≟ False  and point_dist(A_Prepos_l[A_HOR_R],A_Prepos_l[A_VR1])>0.03)
      Folder if move from home
        j_cp := get_actual_joint_positions()
        If b2_left_par removedSiblings(If(type=Else checkContinuously=false, children(Assignment(valueSource=Expression, variable=touch_result, expression=pose_trans(touch_result,p[(Touch_dis-offset_2f_begin)/1000,0,0,0,0,0])))))
          If norm(b_touch_pos[1]*1000)>300
            inner_p := p[-10/1000,-35/1000,0,0,0,0]
          Else 
            inner_p := p[0,0,0,0,0,0]
          j_tp := get_inverse_kin(pose_add(b_touch_pos,inner_p),qnear=left_j)
        Else 
          If norm(b_touch_pos[1]*1000)>300
            inner_p := p[-10/1000,35/1000,0,0,0,0]
          Else 
            inner_p := p[0,0,0,0,0,0]
          j_tp := get_inverse_kin(pose_add(b_touch_pos,inner_p),qnear=right_j)
        Script: j_cp[0]=j_tp[0]
        Script: j_cp[1]=j_cp[1]+(j_tp[1]-j_cp[1])/2
        Script: j_cp[2]=j_cp[2]+(j_tp[2]-j_cp[2])/3
        Script: j_cp[3]=j_cp[3]+(j_tp[3]-j_cp[3])/3
        Script: j_cp[4]=j_cp[4]+(j_tp[4]-j_cp[4])/1
        Script: j_cp[5]=j_cp[5]+(j_tp[5]-j_cp[5])/1
        MoveJ speed 60 deg/s, acceleration 80 deg/s^2 (useActiveTCP=true)
          Waypoint Waypoint (Variable): variable=j_cp
        j_tp := [j_cp[0],j_cp[1],j_cp[2],j_cp[3],j_tp[4],j_tp[5]]
        MoveJ speed 60 deg/s, acceleration 80 deg/s^2 (useActiveTCP=true)
          Waypoint Waypoint (Variable): variable=j_tp
  MoveL speed 350 mm/s, acceleration 350 mm/s^2 (useActiveTCP=true) feature=Base
    Waypoint Waypoint (Variable): variable=b_touch_pos
  SuppressedNode
    MoveL speed 500 mm/s, acceleration 700 mm/s^2 (useActiveTCP=true) feature=Base
      Waypoint Waypoint (Variable): variable=b_touch_pos
  Folder touch_3f_down
    SuppressedNode
      touch_result := touch_fun2(b_touch_pos,b2_left_par,b9_touch_sens)
    touch_result := touch_fun2(b_touch_pos,b2_left_par,b9_touch_sens,b2_par_cd)
    If Scallup_check≟ False
      touch_result := pose_trans(touch_result,p[-(Touch_dis)/1000,0,0,0,0,0])
    Else 
      Scallup_check := False
    SuppressedNode
      touch_result := pose_trans(touch_fun2(b_touch_pos,b2_left_par,b9_touch_sens),p[(-Touch_dis)/1000,0,0,0,0,0])
    SuppressedNode
      touch_result := pose_add(touch_fun2(b_touch_pos,b2_left_par,b9_touch_sens),p[0,0,(-Touch_dis)/1000,0,0,0])
    Script: A_Touch_p[A_sel_v]=touch_result
    If EXT_flag1[3]≟ True
      MoveL speed 150 mm/s, acceleration 300 mm/s^2 (useActiveTCP=true) feature=Base
        manual_tp := tilt_3f_fun(A_Touch_p[A_sel_v],basic_tilt_3f,0)
        manual_tp := pose_trans(manual_tp, p[0,0,-10/1000,0,0,0])
        Waypoint Waypoint (Variable): variable=manual_tp
        Wait Sleep waitTime=1.5
  Folder touch_3f_up [hidden by the author, left out]
  SuppressedNode
    If b2_left_par≟ False removedSiblings(If(type=Else checkContinuously=false, children(Move(motionType=MoveL speed=0.25 acceleration=0.5 useActiveTCP=true, feature=Base, children(Waypoint(type=Fixed name=left_prep_2, position(joints=1.018446445465088, -0.9104264418231409, -1.5978406111346644, -1.808516804371969, 1.480364203453064, 1.670091986656189 pose=0.3993240040399514, 0.30492397897144813, 0.1552705350508301, -2.012034455963345, -1.010425771245131, -1.445571191773495), poseInFeatureCoordinates=poseInFeatureCoordinates, outputFlangePose=[0.171612, 0.04986, 0.428405, -1.197922, 2.476324, 0.179165]))))))
      MoveL speed 250 mm/s, acceleration 500 mm/s^2 (useActiveTCP=true) feature=Base
        Waypoint right_prep_2: TCP in base x=454.066 y=-283.902 z=116.638 mm, rx=2.2253 ry=-0.6942 rz=1.4835 rad; joints [20.297, -58.556, -92.591, -108.708, 71.582, 144.682] deg; flange x=195.53 y=-75.381 z=401.578 mm, rx=0.8644 ry=2.6591 rz=-0.2158 rad
